// TIA Portal V17 export
// export: Created 2023-02-26T22:28:45.699175Z, ExportSetting WithDefaults, DisplayName Totally Integrated Automation Portal, DisplayVersion V17, DisplayName TIA Portal Openness, DisplayVersion V17, DisplayName TIA Portal Version Control Interface, DisplayVersion V17, DisplayName TIA Portal Test Suite Advanced, DisplayVersion V17, DisplayName STEP 7 Professional, DisplayVersion V17, DisplayName SIMATIC Energy Suite, DisplayVersion V17, DisplayName STEP 7 Safety, DisplayVersion V17, DisplayName WinCC Professional, DisplayVersion V17
FUNCTION_BLOCK "ERR_EStop"   // FB6, LAD
{ S7_Optimized_Access := 'TRUE' }
VERSION : 0.1
// stored: AutoNumber true, IsIECCheckEnabled false, IsRetainMemResEnabled false, MemoryReserve 100, SetENOAutomatically false, UDAEnableTagReadback false
   VAR_INPUT
      EStopButton : Bool;
      ResetButton : Bool;
   END_VAR
   VAR_OUTPUT
      Error : Bool;
   END_VAR
   VAR
      P_ResetButton : Bool;
   END_VAR
   VAR_TEMP   // added for the SCL form of the ladder/FBD networks
      _w1 : Bool;
   END_VAR
BEGIN

REGION Network 1
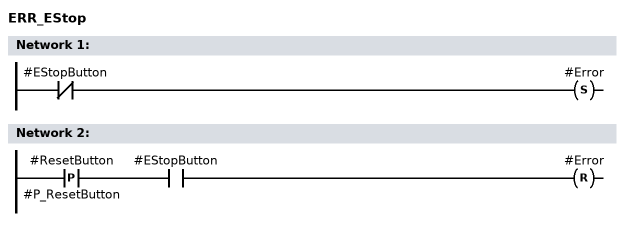
   RUNG wire#powerrail
      I_Contact( #EStopButton )
      S_Coil( #Error )
   END_RUNG
   // the same network as SCL:
   IF NOT #EStopButton THEN #Error := TRUE; END_IF;
END_REGION

REGION Network 2
   RUNG wire#powerrail
      P_Contact(operand := #ResetButton, bit := #P_ResetButton)
      Contact( #EStopButton )
      R_Coil( #Error )
   END_RUNG
   // the same network as SCL:
   #_w1 := #ResetButton AND NOT #P_ResetButton;   // rising edge of #ResetButton
   #P_ResetButton := #ResetButton;
   IF #_w1 AND #EStopButton THEN #Error := FALSE; END_IF;
END_REGION
END_FUNCTION_BLOCK
